TYPE (* IEC61131-3, Table 14#5 *)
  (* Standard: 1131-3 *)
  (* Version 0.0, 1/8/2024, Cheyan, Schneider Electric, Template *)
  PACKAGE Main;
  {SET_ATTRIBUTE(nxtDataType, iTGfw+cvqGRTVq2zQ9VNc0yfo+8yX9MnEbsH95Pdz7/sWlSqSXkpQS5z4aNszWL7dIc+u1teRKZmhRDl9zNqgQ==)}
  stVal : (
    item1,
    item2,
    item3
  );
END_TYPE
